// TIA Portal V18 export
// export: Created 2000-01-01T00:00:00.0000000Z, ExportSetting None
DATA_BLOCK "DB_Motor"   // DB180
{ S7_Optimized_Access := 'FALSE' }
   VAR
      StartCmd : Bool := false;
      StopCmd : Bool := false;
      ResetCmd : Bool := false;
      Fault : Bool := false;
      RunLatch : Bool := false;
      RunFeedback : Bool := false;
      SpeedSetpoint : Real := 0.0;
      SpeedActual : Real := 0.0;
   END_VAR
BEGIN
END_DATA_BLOCK
